# EPICS substitutions: ek9000App/Db/EL3022.substitutions
file EL3022.template
{       pattern
        {
                TERMINAL,

        }
        {
        }
}
